TYPE robot_modes_t :
( 	HM,
	PP,
	CSP
);
END_TYPE

(* stored: Version 1.1.0.1, ProductVersion 3.1.4024.12
   DUT robot_modes_t: Id {ec6bbfac-c85b-4d24-9378-81c105b801c2} *)
